FUNCTION_BLOCK FB_ScaleIN
VAR_INPUT
	inputForScaling : REAL;
	inMin : REAL;
	inMax : REAL;
	outMin : REAL;
	outMax : REAL;
	ctrlCycletime : TIME;
	taskCycletime : TIME;
END_VAR
VAR_OUTPUT
	scaledOutputInt : DINT;
	scaledOutputReal : REAL;
END_VAR
VAR
	fbScale : FB_CTRL_SCALE;
	stParamsForScaling : ST_CTRL_SCALE_PARAMS;
	
END_VAR

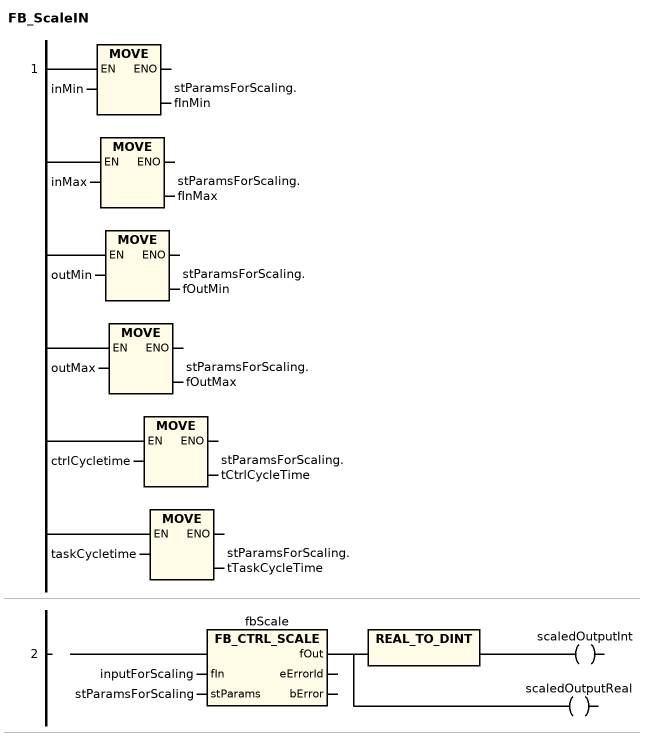
// NETWORK 1
stParamsForScaling.fInMin := inMin;
stParamsForScaling.fInMax := inMax;
stParamsForScaling.fOutMin := outMin;
stParamsForScaling.fOutMax := outMax;
stParamsForScaling.tCtrlCycleTime := ctrlCycletime;
stParamsForScaling.tTaskCycleTime := taskCycletime;

// NETWORK 2
fbScale(fIn := inputForScaling, stParams := stParamsForScaling); // FB_CTRL_SCALE
scaledOutputInt := REAL_TO_DINT(fbScale.fOut);
scaledOutputReal := fbScale.fOut;

END_FUNCTION_BLOCK

(* stored: Version 1.1.0.1, ProductVersion 3.1.4024.13
   POU FB_ScaleIN: Id {7843b705-09b3-45a1-9c1c-f82a96a4ffe4}, SpecialFunc None *)
